FUNCTION_BLOCK FB_PressureMonitor
VAR_IN_OUT
	fbSensors : ARRAY[1..GVL.pressureSensorCount] OF ST_PressureSensor;
END_VAR

VAR
	fbScale : ARRAY[1..GVL.pressureSensorCount] OF FB_ScaleAnalog;
	i : INT;
END_VAR

FOR i := 1 TO GVL.pressureSensorCount DO
	fbScale[i](
		fbRawValue := fbSensors[i].RawValue,
		fbInputMin := fbSensors[i].InputMin,
		fbInputMax := fbSensors[i].InputMax,
		fbOutputMin := fbSensors[i].OutputMin,
		fbOutputMax := fbSensors[i].OutputMax,
		fbScaledValue => fbSensors[i].ScaledValue,
		fbRangeError => fbSensors[i].RangeError);
END_FOR

END_FUNCTION_BLOCK

(* stored: Version 1.1.0.1
   POU FB_PressureMonitor: Id {c3d4e5f6-7a8b-9c0d-1e2f-3a4b5c6d7e8f}, SpecialFunc None *)
